{attribute addProperty BoxType "EL5122-0000-0016"}
{attribute addProperty Id "Enable_latch_extern_on_positive_edgeBIT10.1252Set_counterBIT10.1253Enable_latch_extern_on_negative_edgeBIT10.1254Set_software_gateBIT10.1259Set_counter_on_latch_extern_on_positive_edgeBIT10.12510Set_counter_on_latch_extern_on_negative_edgeBIT10.12511"}
{attribute addProperty CRC "639171011"}
{attribute addProperty SizeInBites "16"}
{attribute addProperty SizeInBytes "2"}
TYPE Control_2618F9C3 :
STRUCT
	{attribute 'hide'}
	reserve_1 : BIT;
	{attribute addProperty Name "Enable_latch_extern_on_positive_edge"}
	Enable_latch_extern_on_positive_edge : BIT;
	{attribute addProperty Name "Set_counter"}
	Set_counter : BIT;
	{attribute addProperty Name "Enable_latch_extern_on_negative_edge"}
	Enable_latch_extern_on_negative_edge : BIT;
	{attribute 'hide'}
	reserve_2_BIT_0 : BIT;
	{attribute 'hide'}
	reserve_2_BIT_1 : BIT;
	{attribute 'hide'}
	reserve_2_BIT_2 : BIT;
	{attribute 'hide'}
	reserve_3 : BIT;
	{attribute addProperty Name "Set_software_gate"}
	Set_software_gate : BIT;
	{attribute addProperty Name "Set_counter_on_latch_extern_on_positive_edge"}
	Set_counter_on_latch_extern_on_positive_edge : BIT;
	{attribute addProperty Name "Set_counter_on_latch_extern_on_negative_edge"}
	Set_counter_on_latch_extern_on_negative_edge : BIT;
	{attribute 'hide'}
	reserve_4 : BIT;
	{attribute 'hide'}
	reserve_5 : BIT;
	{attribute 'hide'}
	reserve_6_BIT_0 : BIT;
	{attribute 'hide'}
	reserve_6_BIT_1 : BIT;
	{attribute 'hide'}
	reserve_6_BIT_2 : BIT;
END_STRUCT
END_TYPE

(* stored: Version 1.2.0.0, ProductVersion 3.1.4024.9
   DUT Control_2618F9C3: Id {e7838dff-8b40-414c-8e25-ccedb6be9a17} *)
